DATA_BLOCK "StatusDB"
{ S7_Optimized_Access := 'TRUE' }
VERSION : '1.0'
UNLINKED
NON_RETAIN
VAR
    CURRENT_STATUS : "Status_001";
    STATUS_HISTORY : ARRAY[0..99] OF "Status_001";
    LAST_ERROR_MESSAGE : STRING;
END_VAR
END_DATA_BLOCK